DATA_BLOCK "ST10_FB_Tower_4Lamp_DB"
VAR
  TON : Array[0..10] of TON_TIME;
  sRed_Lamp : Bool;
  sResetButtonPressed : Bool;
  sBuzzerOnCurrentVal : Int;
  P_TRIG : Array[0..10] of Bool;
  N_TRIG : Array[0..10] of Bool;
END_VAR
BEGIN
END_DATA_BLOCK
